FUNCTION_BLOCK FB_StaticHandler_n EXTENDS FB_BaseHandler
VAR_INPUT
END_VAR
VAR_OUTPUT
END_VAR
VAR
END_VAR

METHOD handle : BOOL
VAR_INPUT
	request	:	STRING;
END_VAR
ADSLOGSTR(ADSLOG_MSGTYPE_MSGBOX, request , '');
END_METHOD

END_FUNCTION_BLOCK

(* stored: Version 1.1.0.1, ProductVersion 3.1.4024.12
   POU FB_StaticHandler_n: Id {b27f75cc-7db2-0c1d-126c-3d51b98cb138}, SpecialFunc None
   Method handle: Id {8651466d-3bb6-025a-09d9-ba8112cfecf5} *)
